// TIA Portal V19 export
VAR_GLOBAL   // PLC tag table "U2Em1_Output"
   requestTrayDelivery_standalone_U2EM1 AT %Q30042.0 : Bool;   // 单机请求出
   vfdBusy_standalone_U2EM1 AT %Q30042.1 : Bool;   // 单机出料中
   Received_the_shipment_in_place_U2EM1 AT %Q30042.2 : Bool;   // 单机收到物料
   emAlarm_standalone_U2EM1 AT %Q30042.3 : Bool;   // 单机异常
   Tray_waiting_to_be_released_U2EM1 AT %Q30042.4 : Bool;   // 单机有托盘待出
   Allow_logistics_lines_to_exit_U2EM1 AT %Q30043.0 : Bool;   // 单机允许物流线出
   Notify_the_logistics_line_to_arrive_in_place_U2EM1 AT %Q30043.1 : Bool;   // 单机通知物流线出到位
   Single_machine_output_in_place_signal_U2EM1 AT %Q30043.2 : Bool;   // 单机收到物流线收到的单机出到位信号
   idle_standalone_U2EM1 AT %Q30043.3 : Bool;   // 单机空闲
END_VAR
